		IF bBeendet OR bReset THEN
			bReset := FALSE;
			SFCReset := FALSE;
			iState := 0;
		END_IF
	2: // ABGESCHLOSSEN
		IF SFCCurrentStep = 'Init' THEN
			iState := 0;
		END_IF
END_CASE

ACTION ACT_1:
R_Move.P_RobotParam := RobParam[0];
END_ACTION

ACTION ACT_2:
R_Move.P_RobotParam := RobParam[1];
END_ACTION

ACTION ACT_3:
R_Move.P_RobotParam := RobParam[2];
R_Move.P_Erreicht := ErreichtParam;
END_ACTION

ACTION ACT_4:
R_Move.P_RobotParam := RobParam[3];
END_ACTION

ACTION ACT_5:
R_Move.P_RobotParam := RobParam[4];
END_ACTION

ACTION ACT_Ablauf:
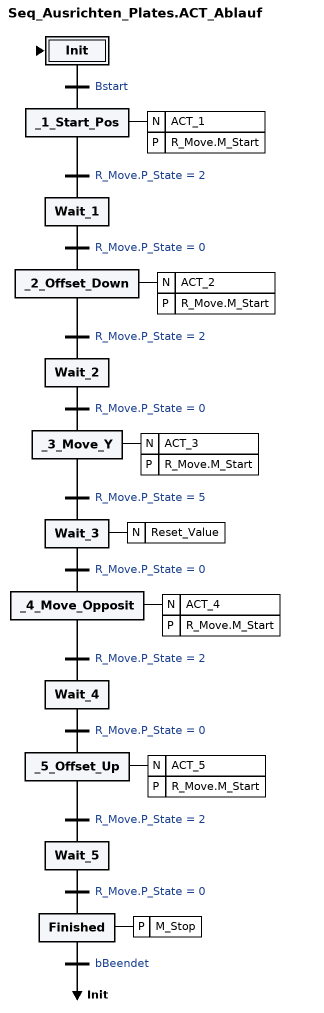
INITIAL_STEP Init:
END_STEP
TRANSITION FROM Init TO _1_Start_Pos
    := Bstart;
END_TRANSITION
STEP _1_Start_Pos:
    ACT_1(N);
    R_Move.M_Start(P);
END_STEP
TRANSITION FROM _1_Start_Pos TO Wait_1
    := R_Move.P_State = 2;
END_TRANSITION
STEP Wait_1:
END_STEP
TRANSITION FROM Wait_1 TO _2_Offset_Down
    := R_Move.P_State = 0;
END_TRANSITION
STEP _2_Offset_Down:
    ACT_2(N);
    R_Move.M_Start(P);
END_STEP
TRANSITION FROM _2_Offset_Down TO Wait_2
    := R_Move.P_State = 2;
END_TRANSITION
STEP Wait_2:
END_STEP
TRANSITION FROM Wait_2 TO _3_Move_Y
    := R_Move.P_State = 0;
END_TRANSITION
STEP _3_Move_Y:
    ACT_3(N);
    R_Move.M_Start(P);
END_STEP
TRANSITION FROM _3_Move_Y TO Wait_3
    := R_Move.P_State = 5;
END_TRANSITION
STEP Wait_3:
    Reset_Value(N);
END_STEP
TRANSITION FROM Wait_3 TO _4_Move_Opposit
    := R_Move.P_State = 0;
END_TRANSITION
STEP _4_Move_Opposit:
    ACT_4(N);
    R_Move.M_Start(P);
END_STEP
TRANSITION FROM _4_Move_Opposit TO Wait_4
    := R_Move.P_State = 2;
END_TRANSITION
STEP Wait_4:
END_STEP
TRANSITION FROM Wait_4 TO _5_Offset_Up
    := R_Move.P_State = 0;
END_TRANSITION
STEP _5_Offset_Up:
    ACT_5(N);
    R_Move.M_Start(P);
END_STEP
TRANSITION FROM _5_Offset_Up TO Wait_5
    := R_Move.P_State = 2;
END_TRANSITION
STEP Wait_5:
END_STEP
TRANSITION FROM Wait_5 TO Finished
    := R_Move.P_State = 0;
END_TRANSITION
STEP Finished:
    M_Stop(P);
END_STEP
TRANSITION FROM Finished TO Init
    := bBeendet;
END_TRANSITION
END_ACTION

ACTION Reset_Value:
ErreichtParamReset.Fx := 0;
ErreichtParamReset.Fy := 0;
ErreichtParamReset.Fz := 0;

R_Move.P_Erreicht := ErreichtParamReset;
END_ACTION

END_FUNCTION_BLOCK

// ---- POUs/01_Prozessmodell/02_Sequenzen/01_Version_1/Seq_Get_Part.TcPOU
FUNCTION_BLOCK Seq_Get_Part EXTENDS FB_Basis IMPLEMENTS I_Sequenz
VAR_INPUT
	// Skillzuweisung
	R_Move					:I_Skill_Roboter;
	G_Move					:I_Skill_SmartGreifer;
	
	// Prozessparameter		
	RobParam				:ARRAY[0..2] OF sRoboterProzessVariablen;
	GripParam				:ARRAY[0..1] OF sSmartGreiferProzessVariablen;
END_VAR
VAR_OUTPUT
END_VAR
VAR
	// Interne Sequenzen
	Seq_Ausrichten			:Seq_Ausrichten;
END_VAR

// Ablauf
ACT_Ablauf();

// Zustandshandling
CASE iState OF
	0:	// BEREIT
		IF bStart THEN
			iState := 1;
		END_IF
	1:	// LAUFEND
		IF eSysCommand = 4 THEN
			bReset := TRUE;
			SFCReset := TRUE;
		END_IF
		
		IF bBeendet OR bReset THEN
			bReset := FALSE;
			SFCReset := FALSE;
			iState := 0;
		END_IF
	2: // ABGESCHLOSSEN
		IF SFCCurrentStep = 'Init' THEN
			iState := 0;
		END_IF
END_CASE

ACTION ACT_Ablauf:
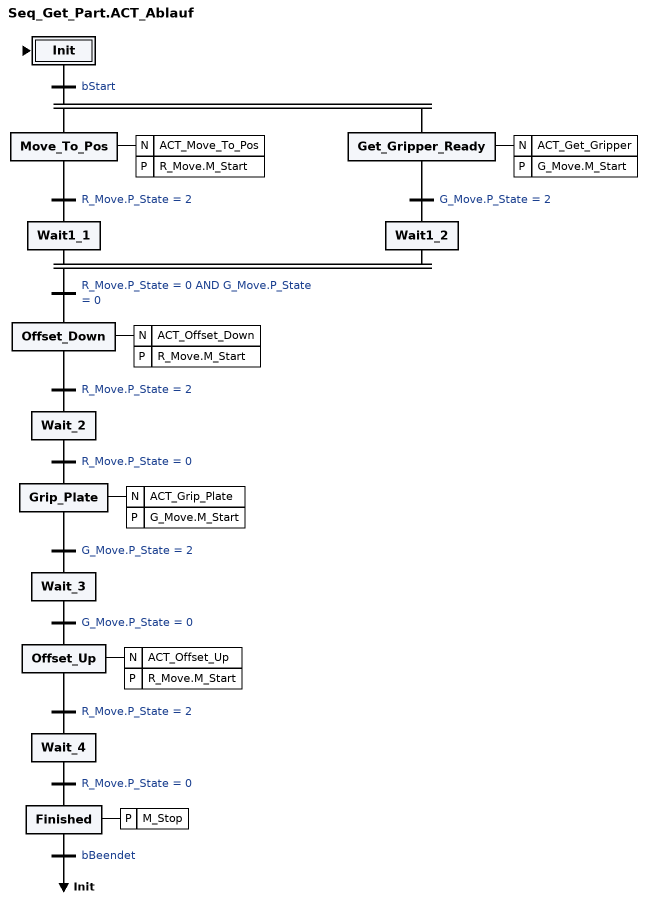
INITIAL_STEP Init:
END_STEP
TRANSITION FROM Init TO (Move_To_Pos, Get_Gripper_Ready)
    := bStart;
END_TRANSITION
STEP Move_To_Pos:
    ACT_Move_To_Pos(N);
    R_Move.M_Start(P);
END_STEP
TRANSITION FROM Move_To_Pos TO Wait1_1
    := R_Move.P_State = 2;
END_TRANSITION
STEP Wait1_1:
END_STEP
STEP Get_Gripper_Ready:
    ACT_Get_Gripper(N);
    G_Move.M_Start(P);
END_STEP
TRANSITION FROM Get_Gripper_Ready TO Wait1_2
    := G_Move.P_State = 2;
END_TRANSITION
STEP Wait1_2:
END_STEP
TRANSITION FROM (Wait1_1, Wait1_2) TO Offset_Down
    := R_Move.P_State = 0 AND G_Move.P_State = 0;
END_TRANSITION
STEP Offset_Down:
    ACT_Offset_Down(N);
    R_Move.M_Start(P);
END_STEP
TRANSITION FROM Offset_Down TO Wait_2
    := R_Move.P_State = 2;
END_TRANSITION
STEP Wait_2:
END_STEP
TRANSITION FROM Wait_2 TO Grip_Plate
    := R_Move.P_State = 0;
END_TRANSITION
STEP Grip_Plate:
    ACT_Grip_Plate(N);
    G_Move.M_Start(P);
END_STEP
TRANSITION FROM Grip_Plate TO Wait_3
    := G_Move.P_State = 2;
END_TRANSITION
STEP Wait_3:
END_STEP
TRANSITION FROM Wait_3 TO Offset_Up
    := G_Move.P_State = 0;
END_TRANSITION
STEP Offset_Up:
    ACT_Offset_Up(N);
    R_Move.M_Start(P);
END_STEP
TRANSITION FROM Offset_Up TO Wait_4
    := R_Move.P_State = 2;
END_TRANSITION
STEP Wait_4:
END_STEP
TRANSITION FROM Wait_4 TO Finished
    := R_Move.P_State = 0;
END_TRANSITION
STEP Finished:
    M_Stop(P);
END_STEP
TRANSITION FROM Finished TO Init
    := bBeendet;
END_TRANSITION
END_ACTION

ACTION ACT_Get_Gripper:
G_Move.P_SGripperParam := GripParam[0];
END_ACTION

ACTION ACT_Grip_Plate:
G_Move.P_SGripperParam := GripParam[1];
END_ACTION

ACTION ACT_Move_To_Pos:
R_Move.P_RobotParam := RobParam[0];
END_ACTION

ACTION ACT_Offset_Down:
R_Move.P_RobotParam := RobParam[1];
END_ACTION

ACTION ACT_Offset_Up:
R_Move.P_RobotParam := RobParam[2];
END_ACTION

END_FUNCTION_BLOCK

// ---- POUs/01_Prozessmodell/02_Sequenzen/01_Version_1/Seq_Set_MPlate.TcPOU
FUNCTION_BLOCK Seq_Set_MPlate EXTENDS FB_Basis IMPLEMENTS I_Sequenz
VAR_INPUT
	// Skillzuweisung
	R_Move			:I_Skill_RoboterErweitert;
	G_Move			:I_Skill_SmartGreifer; 
	
	// Prozessparameter		
	RobParam				:ARRAY[0..2] OF sRoboterProzessVariablen;
	GripParam				:sSmartGreiferProzessVariablen;
	ErreichtParam			:sKraftVariablen;
END_VAR
VAR_OUTPUT
END_VAR
VAR
	ErreichtParamReset		:sKraftVariablen;
END_VAR

// Ablauf
ACT_Ablauf();

// Zustandshandling
CASE iState OF
	0:	// BEREIT
		IF bStart THEN
			iState := 1;
		END_IF
	1:	// LAUFEND
		IF eSysCommand = 4 THEN
			bReset := TRUE;
			SFCReset := TRUE;
		END_IF
		
		IF bBeendet OR bReset THEN
			bReset := FALSE;
			SFCReset := FALSE;
			iState := 0;
		END_IF
	2: // ABGESCHLOSSEN
		IF SFCCurrentStep = 'Init' THEN
			iState := 0;
		END_IF
END_CASE

ACTION ACT_1:
R_Move.P_RobotParam := RobParam[0];
END_ACTION

ACTION ACT_2:
R_Move.P_RobotParam := RobParam[1];
R_Move.P_Erreicht := ErreichtParam;
END_ACTION

ACTION ACT_3:
G_Move.P_SGripperParam := GripParam;
END_ACTION

ACTION ACT_4:
R_Move.P_RobotParam := RobParam[2];
END_ACTION

ACTION ACT_Ablauf:
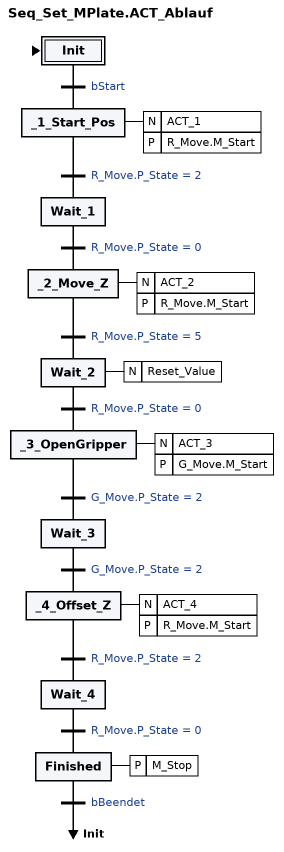
INITIAL_STEP Init:
END_STEP
TRANSITION FROM Init TO _1_Start_Pos
    := bStart;
END_TRANSITION
STEP _1_Start_Pos:
    ACT_1(N);
    R_Move.M_Start(P);
END_STEP
TRANSITION FROM _1_Start_Pos TO Wait_1
    := R_Move.P_State = 2;
END_TRANSITION
STEP Wait_1:
END_STEP
TRANSITION FROM Wait_1 TO _2_Move_Z
    := R_Move.P_State = 0;
END_TRANSITION
STEP _2_Move_Z:
    ACT_2(N);
    R_Move.M_Start(P);
END_STEP
TRANSITION FROM _2_Move_Z TO Wait_2
    := R_Move.P_State = 5;
END_TRANSITION
STEP Wait_2:
    Reset_Value(N);
END_STEP
TRANSITION FROM Wait_2 TO _3_OpenGripper
    := R_Move.P_State = 0;
END_TRANSITION
STEP _3_OpenGripper:
    ACT_3(N);
    G_Move.M_Start(P);
END_STEP
TRANSITION FROM _3_OpenGripper TO Wait_3
    := G_Move.P_State = 2;
END_TRANSITION
STEP Wait_3:
END_STEP
TRANSITION FROM Wait_3 TO _4_Offset_Z
    := G_Move.P_State = 2;
END_TRANSITION
STEP _4_Offset_Z:
    ACT_4(N);
    R_Move.M_Start(P);
END_STEP
TRANSITION FROM _4_Offset_Z TO Wait_4
    := R_Move.P_State = 2;
END_TRANSITION
STEP Wait_4:
END_STEP
TRANSITION FROM Wait_4 TO Finished
    := R_Move.P_State = 0;
END_TRANSITION
STEP Finished:
    M_Stop(P);
END_STEP
TRANSITION FROM Finished TO Init
    := bBeendet;
END_TRANSITION
END_ACTION

ACTION Reset_Value:
ErreichtParamReset.Fx := 0;
ErreichtParamReset.Fy := 0;
ErreichtParamReset.Fz := 0;

R_Move.P_Erreicht := ErreichtParamReset;
END_ACTION

END_FUNCTION_BLOCK

// ---- POUs/01_Prozessmodell/03_Arbeitsplan/AP_V1.TcPOU
PROGRAM AP_V1
VAR
	GetPlate			:Seq_Get_Part;
	SetPlate1			:Seq_Set_Plate_1;
	SetPlate2			:Seq_Set_Plate_2;
	AusrichtenPlates 	:Seq_Ausrichten_Plates;
	SetMountingPlate	:Seq_Set_MPlate;
	AusrichtenMP		:Seq_Ausrichten_MPlate;
END_VAR

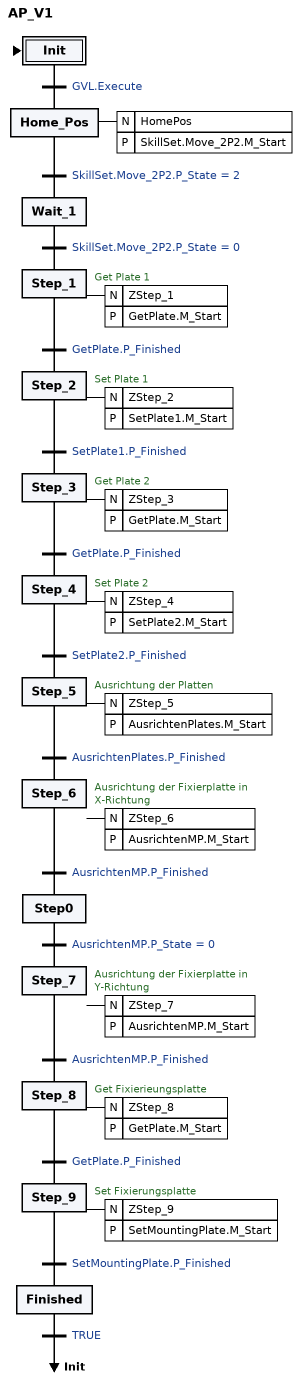
INITIAL_STEP Init:
END_STEP
TRANSITION FROM Init TO Home_Pos
    := GVL.Execute;
END_TRANSITION
STEP Home_Pos:
    HomePos(N);
    SkillSet.Move_2P2.M_Start(P);
END_STEP
TRANSITION FROM Home_Pos TO Wait_1
    := SkillSet.Move_2P2.P_State = 2;
END_TRANSITION
STEP Wait_1:
END_STEP
TRANSITION FROM Wait_1 TO Step_1
    := SkillSet.Move_2P2.P_State = 0;
END_TRANSITION
// Get Plate 1
STEP Step_1:
    ZStep_1(N);
    GetPlate.M_Start(P);
END_STEP
TRANSITION FROM Step_1 TO Step_2
    := GetPlate.P_Finished;
END_TRANSITION
// Set Plate 1
STEP Step_2:
    ZStep_2(N);
    SetPlate1.M_Start(P);
END_STEP
TRANSITION FROM Step_2 TO Step_3
    := SetPlate1.P_Finished;
END_TRANSITION
// Get Plate 2
STEP Step_3:
    ZStep_3(N);
    GetPlate.M_Start(P);
END_STEP
TRANSITION FROM Step_3 TO Step_4
    := GetPlate.P_Finished;
END_TRANSITION
// Set Plate 2
STEP Step_4:
    ZStep_4(N);
    SetPlate2.M_Start(P);
END_STEP
TRANSITION FROM Step_4 TO Step_5
    := SetPlate2.P_Finished;
END_TRANSITION
// Ausrichtung der Platten
STEP Step_5:
    ZStep_5(N);
    AusrichtenPlates.M_Start(P);
END_STEP
TRANSITION FROM Step_5 TO Step_6
    := AusrichtenPlates.P_Finished;
END_TRANSITION
// Ausrichtung der Fixierplatte in X-Richtung
STEP Step_6:
    ZStep_6(N);
    AusrichtenMP.M_Start(P);
END_STEP
TRANSITION FROM Step_6 TO Step0
    := AusrichtenMP.P_Finished;
END_TRANSITION
STEP Step0:
END_STEP
TRANSITION FROM Step0 TO Step_7
    := AusrichtenMP.P_State = 0;
END_TRANSITION
// Ausrichtung der Fixierplatte in Y-Richtung
STEP Step_7:
    ZStep_7(N);
    AusrichtenMP.M_Start(P);
END_STEP
TRANSITION FROM Step_7 TO Step_8
    := AusrichtenMP.P_Finished;
END_TRANSITION
// Get Fixierieungsplatte
STEP Step_8:
    ZStep_8(N);
    GetPlate.M_Start(P);
END_STEP
TRANSITION FROM Step_8 TO Step_9
    := GetPlate.P_Finished;
END_TRANSITION
// Set Fixierungsplatte
STEP Step_9:
    ZStep_9(N);
    SetMountingPlate.M_Start(P);
END_STEP
TRANSITION FROM Step_9 TO Finished
    := SetMountingPlate.P_Finished;
END_TRANSITION
STEP Finished:
END_STEP
TRANSITION FROM Finished TO Init
    := TRUE;
END_TRANSITION

ACTION HomePos:
SkillSet.Move_2P2.P_RobotParam := PunkteZuweisung_Temp.PHome;
END_ACTION

ACTION ZStep_1:
GetPlate(
    eSysCommand := GVL.SystemCommand,
    R_Move := SkillSet.Move_2P2,
    G_Move := SkillSet.Grip_2P2,
    RobParam := PunkteZuweisung_Temp.R_Data_1,
    GripParam := PunkteZuweisung_Temp.G_Data_1); // Seq_Get_Part
END_ACTION

ACTION ZStep_2:
SetPlate1(
    eSysCommand := GVL.SystemCommand,
    R_Move := SkillSet.Move_2P2_Advanced,
    G_Move := SkillSet.Grip_2P2,
    RobParam := PunkteZuweisung_Temp.R_Data_2,
    GripParam := PunkteZuweisung_Temp.Plate_Open,
    ErreichtParam := PunkteZuweisung_Temp.S_Data_1); // Seq_Set_Plate_1
END_ACTION

ACTION ZStep_3:
GetPlate(
    eSysCommand := GVL.SystemCommand,
    R_Move := SkillSet.Move_2P2,
    G_Move := SkillSet.Grip_2P2,
    RobParam := PunkteZuweisung_Temp.R_Data_3,
    GripParam := PunkteZuweisung_Temp.G_Data_1); // Seq_Get_Part
END_ACTION

ACTION ZStep_4:
SetPlate2(
    eSysCommand := GVL.SystemCommand,
    R_Move := SkillSet.Move_2P2_Advanced,
    G_Move := SkillSet.Grip_2P2,
    RobParam := PunkteZuweisung_Temp.R_Data_4,
    GripParam := PunkteZuweisung_Temp.Plate_Open,
    ErreichtParam := PunkteZuweisung_Temp.AnstossX); // Seq_Set_Plate_2
END_ACTION

ACTION ZStep_5:
AusrichtenPlates(
    eSysCommand := GVL.SystemCommand,
    R_Move := SkillSet.Move_2P2_Advanced,
    RobParam := PunkteZuweisung_Temp.R_Data_5,
    ErreichtParam := PunkteZuweisung_Temp.AnstossX); // Seq_Ausrichten_Plates
END_ACTION

ACTION ZStep_6:
AusrichtenMP(
    eSysCommand := GVL.SystemCommand,
    R_Move := SkillSet.Move_2P2_Advanced,
    G_Move := SkillSet.Grip_2P2,
    RobParam := PunkteZuweisung_Temp.R_Data_6,
    ErreichtParam := PunkteZuweisung_Temp.AnstossnX,
    GripParam := PunkteZuweisung_Temp.GripperClossed); // Seq_Ausrichten_MPlate
END_ACTION

ACTION ZStep_7:
AusrichtenMP(
    eSysCommand := GVL.SystemCommand,
    R_Move := SkillSet.Move_2P2_Advanced,
    G_Move := SkillSet.Grip_2P2,
    RobParam := PunkteZuweisung_Temp.R_Data_7,
    ErreichtParam := PunkteZuweisung_Temp.AnstossnY,
    GripParam := PunkteZuweisung_Temp.GripperClossed); // Seq_Ausrichten_MPlate
END_ACTION

ACTION ZStep_8:
GetPlate(
    eSysCommand := GVl.SystemCommand,
    R_Move := SkillSet.Move_2P2,
    G_Move := Skillset.Grip_2P2,
    RobParam := PunkteZuweisung_Temp.R_Data_8,
    GripParam := PunkteZuweisung_Temp.G_Data_2); // Seq_Get_Part
END_ACTION

ACTION ZStep_9:
SetMountingPlate(
    eSysCommand := GVL.SystemCommand,
    R_Move := SkillSet.Move_2P2_Advanced,
    G_Move := SkillSet.Grip_2P2,
    RobParam := PunkteZuweisung_Temp.R_Data_9,
    GripParam := PunkteZuweisung_Temp.FixPlate_Open,
    ErreichtParam := PunkteZuweisung_Temp.AnstossZ); // Seq_Set_MPlate
END_ACTION

END_PROGRAM

// ---- POUs/01_Prozessmodell/03_Arbeitsplan/AP_V2_1.TcPOU
PROGRAM AP_V2_1
VAR
	// Bedienparameter
	
	// Prozessparameter
	
	// Skill-Instanziierung
	Skill_R_P2P			:Skill_Position_anfahren;
	Skill_R_Ausrichten	:Skill_Position_anfahren_erweitert;
	Skill_G_P2P			:Skill_Greifer_Pos_Anfahren;
	
	// Sequenz-Instanziierung
	Seq_Get_Teil		:Seq_Teile_Hohlen;
	
	
END_VAR

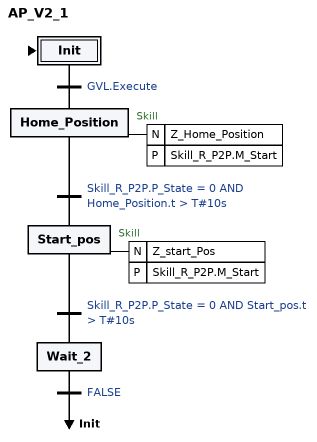
INITIAL_STEP Init:
END_STEP
TRANSITION FROM Init TO Home_Position
    := GVL.Execute;
END_TRANSITION
// Skill
STEP Home_Position:
    Z_Home_Position(N);
    Skill_R_P2P.M_Start(P);
END_STEP
TRANSITION FROM Home_Position TO Start_pos
    := Skill_R_P2P.P_State = 0 AND Home_Position.t > T#10s;
END_TRANSITION
// Skill
STEP Start_pos:
    Z_start_Pos(N);
    Skill_R_P2P.M_Start(P);
END_STEP
TRANSITION FROM Start_pos TO Wait_2
    := Skill_R_P2P.P_State = 0 AND Start_pos.t > T#10s;
END_TRANSITION
STEP Wait_2:
END_STEP
TRANSITION FROM Wait_2 TO Init
    := FALSE;
END_TRANSITION

ACTION Z_Home_Position:
// Skillaufruf
Skill_R_P2P(eSysCommand := GVL.SystemCommand,
			eSysState := GVL.SystemState,
			Objekt := Anlage.UR5,
			iErrorID => GVL.ErrorID);

// Parameterzuweisung
Skill_R_P2P.P_RobotParam := PunkteZuweisung_Temp.PHome;
END_ACTION

ACTION Z_Start_Pos:
// Skillaufruf
Skill_R_P2P(eSysCommand := GVL.SystemCommand,
			eSysState := GVL.SystemState,
			Objekt := Anlage.UR5,
			iErrorID => GVL.ErrorID);

		
// Parameterzuweisung	
Skill_R_P2P.P_RobotParam := PunkteZuweisung_Temp.PGetPlate1;
END_ACTION

END_PROGRAM

// ---- POUs/02_Anlagenmodell/01_Objektklassen/00_Referenz/Basis_Objekt.TcPOU
FUNCTION_BLOCK Basis_Objekt IMPLEMENTS I_Objekt_Roboter
VAR_INPUT
	eSysState			:eSystemState;		// Information über Stand von System
	eSysCommand		  	:eSystemCommand;	// Steuerungsvariabel von System
	iMode				:INT;				// Information über aktuellen Betriebsmodi 
END_VAR
VAR_OUTPUT
	iErrorID			:INT;				// Information um welchen Fehler es sich handelt	
END_VAR
VAR
	iState				:eObjectAktorState;		// Information über Zustand von Skill
	
	// Zustandsvariablen
	bEinschalten			:BOOL;			// Objekt einschalten
	bAusschalten			:BOOL;			// Objekt ausschalten
 	bStarten				:BOOL;			// Objekt starten
	bObjektFertig			:BOOL;			// Objekt hat Prozess abgeschlossen
	bSkillFertig			:BOOL;			// Skill hat Prozess abgeschlossen
	bStoppen				:BOOL;			// Objekt wurde gestoppt
	bResettenSkill			:BOOL;			// Das Objekt wird durch den Skill resettet
	bResettenSystem			:BOOL;			// Das Objekt wird durch das System resettet 
	bFehler					:BOOL;			// Das Objket hat einen Fehler
	
	iFehlerID				:UDINT;

END_VAR

// Instanziierungen
	
//____________________________________________________________________________________________
// Input-Command-Verwaltung
	// System
	IF eSysCommand = 2 AND iState = 0 THEN			// Objekt einschalten
		bEinschalten := TRUE;
	ELSE 
		bEinschalten := FALSE;
	END_IF
	
	IF eSysCommand = 1 AND iState = 1 THEN			// Objekt ausschalten
		bAusschalten := TRUE;		
	ELSE 
		bAusschalten := FALSE;		
	END_IF
	
	IF eSysCommand = 3 THEN							// Objekt beendet Prozess
		bStoppen := TRUE;
	ELSE
		bStoppen := FALSE;
	END_IF
	
	IF eSysCommand = 4 THEN							// System resettet Objekt
		bResettenSystem := TRUE;
	ELSE
		bResettenSystem := FALSE;
	END_IF

//____________________________________________________________________________________________
// Interner Methodenaufruf (Durch System oder Skill)

//____________________________________________________________________________________________
// Datenerfassungsprozess

//____________________________________________________________________________________________
// Zustandsmanagement

IF bFehler THEN 
	iState := 7;
END_IF

CASE iState OF 
	0: // AUS
		// DO
		
		// TRANSITION
			IF bEinschalten THEN																	// Verbindung wird aufgebaut
				iState := 1;
			END_IF
			
	//____________________________________________________________________________________________
	1: // BEREIT
		// DO

		// TRANSITION
																									// Manuell-Modus wird eingeschalten
													
			 IF bStarten THEN																		// Objekt führt Prozessdurch
				 bStarten := FALSE;
				 iState := 3;
			 END_IF			
	//____________________________________________________________________________________________
	2: // MANUELL
		// DO
		
		// TRANSITION
	
	//____________________________________________________________________________________________
	3: // LAUFEND
		// DO
		
		// TRANSITION
			IF bObjektFertig THEN
				bObjektFertig := FALSE;
				iState := 4;
			END_IF
			
			IF bStoppen THEN	
				
				IF bSkillFertig THEN
					bSkillFertig := FALSE;
					iState := 5;
				END_IF
					
				IF bStoppen THEN
					iState := 6;
				END_IF
					
			END_IF
	
	//____________________________________________________________________________________________
	4: // ABGESCHLOSSEN_INTERN
		// DO
		
		// TRANSITION
			IF bResettenSkill THEN																	// Objekt resetten		
				bResettenSkill := FALSE;
				iState := 1;
			END_IF
	//____________________________________________________________________________________________
	5: // ABGESCHLOSSEN_EXTERN
		// DO																					
		
		// TRANSITION
			IF bResettenSkill THEN																	// Objekt resetten
				bResettenSkill := FALSE;
				iState := 1;
			END_IF
	
	//____________________________________________________________________________________________
	6: // GESTOPPT
		// DO
		
		// TRANSITION
			IF bResettenSystem THEN																	// Objekt resetten
				iState := 1;
			END_IF
	
	//____________________________________________________________________________________________
	7: // FEHLER
		// DO
			
		// TRANSITION
			IF bResettenSystem THEN																	// Objekt resetten
				bFehler	 := FALSE;
				iState := 1;
			END_IF
	
END_CASE

METHOD M_Reset : BOOL

bResettenSkill := TRUE;

IF bResettenSkill THEN
	M_Reset := TRUE;
ELSE
	M_Reset := FALSE;
END_IF
END_METHOD

METHOD M_Start : BOOL

// Prüfen von Bedingungen
	// Ist das  System im korrekten Status
	IF eSysState = 1 THEN
		// Ist das Objekt im korrekten Status 
		IF iState = 0 THEN
			bStarten := TRUE;
		END_IF
	END_IF

IF bStarten THEN
	M_Start := TRUE;
ELSE
	M_Start := FALSE;
END_IF
END_METHOD

METHOD M_Stop : BOOL

// Ist das Objekt im korrekten Status 
IF iState = 3 THEN
	bStoppen := TRUE;
END_IF

IF bStoppen THEN
	M_Stop := TRUE;
ELSE
	M_Stop := FALSE;
END_IF
END_METHOD

PROPERTY P_Prozessparameter : sRoboterProzessVariablen
SET
END_SET
END_PROPERTY

PROPERTY P_State : eObjectAktorState
GET
P_State := iState;
END_GET
END_PROPERTY

END_FUNCTION_BLOCK

// ---- POUs/02_Anlagenmodell/01_Objektklassen/00_Referenz/FB_Basis_Objekt_Sensor.TcPOU
FUNCTION_BLOCK FB_Basis_Objekt_Sensor
VAR_INPUT
END_VAR
VAR_OUTPUT
END_VAR
VAR
END_VAR

END_FUNCTION_BLOCK

// ---- GlobalTextList.TcGTLO
TEXTLIST GlobalTextList
  142 = '%'
  560 = '%s'
  874 = 'AUSCHALTEN'
  468 = 'EINSCHALTEN'
  683 = 'Fahren'
  769 = 'Geschwindigkeit:'
  47 = 'Gripper'
  764 = 'KEINE'
  756 = 'Kraft:'
  713 = 'Lesen'
  304 = 'mm'
  839 = 'Position:'
  303 = 'RESETTEN'
  281 = 'START'
  351 = 'STOPPEN'
  785 = 'SystemCommand'
END_TEXTLIST

// ---- VISUs/Visualization.TcVIS
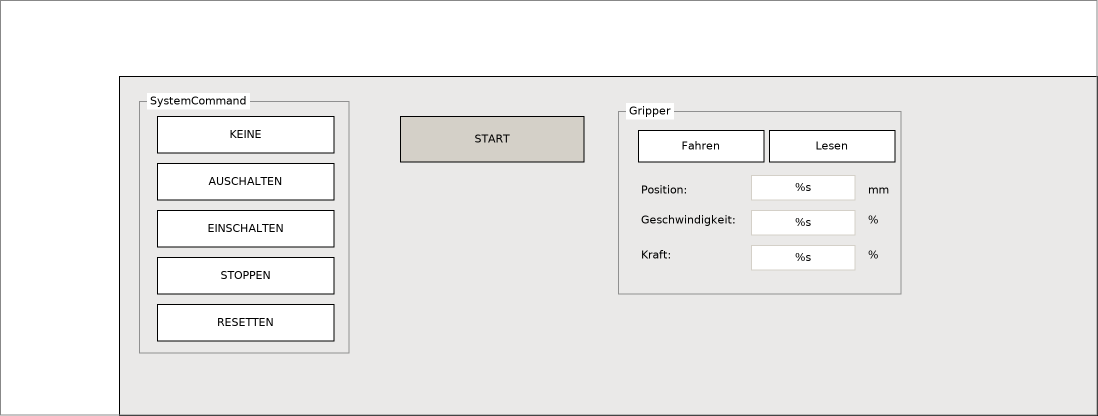
VISUALIZATION Visualization  // 1098x416
VAR_IN_OUT
	
END_VAR

VAR
	iPos		:BYTE;
	iGeschw		:BYTE;
	iKraft		:BYTE;
END_VAR
    Rectangle (119,76 979x340)
    RoundedRectangle (400,116 184x46), "START"
        tap GVL.Execute
    GroupBox (139,93 210x260), "SystemCommand"
        RoundedRectangle (18,70 177x37), "AUSCHALTEN"
            OnMouseClick: execute { GVL.SystemCommand := 1; }
        RoundedRectangle (18,117 177x37), "EINSCHALTEN"
            OnMouseClick: execute { GVL.SystemCommand := 2; }
        RoundedRectangle (18,164 177x37), "STOPPEN"
            OnMouseClick: execute { GVL.SystemCommand := 3; }
        RoundedRectangle (18,211 177x37), "RESETTEN"
            OnMouseClick: execute { GVL.SystemCommand := 4; }
        RoundedRectangle (18,23 177x37), "KEINE"
            OnMouseClick: execute { GVL.SystemCommand := 0; }
    GroupBox (618,103 283x191), "Gripper"
        RoundedRectangle (20,27 126x32), "Fahren"
            OnMouseClick: execute { Anlage.Gripper.M_PositionAnfahren(iPos := iPos, iGeschw := iGeschw, iKraft := iKraft); }
        Textfield (133,72 104x25), "%s", text variable: iPos
            OnMouseDown: write iPos via Edit, format %s
        Textfield (133,107 104x25), "%s", text variable: iGeschw
            OnMouseClick: write iGeschw via Edit, format %d
        Textfield (133,142 104x25), "%s", text variable: iKraft
            OnMouseClick: write iKraft via Edit, format %s
        Label (20,72 95x30), "Position:"
        Label (20,102 95x30), "Geschwindigkeit:"
        Label (20,137 95x30), "Kraft:"
        Label (247,72 30x30), "mm"
        Label (247,102 30x30), "%"
        Label (247,137 25x30), "%"
        RoundedRectangle (151,27 126x32), "Lesen"
            OnMouseClick: execute { Anlage.Gripper.M_StatusLesen(NrOfReg := 3); }
END_VISUALIZATION
